// TIA Portal V18 export
TYPE "KukaRobot_UserOutput_3"
   STRUCT
      Public : Struct
         GO_CurrentMode : USInt;
         GO_CurrentPartType : USInt;
         GO_SpeedActual : USInt;   // Robot speed
         GO_RobotTaskSequence : Byte;
         GO5_RobGrip1Status : Byte;   // Gripper 1 status
         GO6_RobGrip2Status : Byte;   // Gripper 2 state
         GO7_Pallet1Count : Byte;
         GO8_UnloadingPalletCount : Byte;   // Pallet finished product count
         GO9 : Byte;
         GO10 : Byte;
      END_STRUCT;
      Gripper : Struct
         DO129_Grip1GoWork : Bool;   // Clamp 1 goes to work position
         DO130_Grip1GoHome : Bool;   // Clamp 1 to original position
         DO131_Grip2GoWork : Bool;   // Clamp 2 goes to work position
         DO132_Grip2GoHome : Bool;   // Clamp 2 to original position
         DO133 : Bool;
         DO134 : Bool;
         DO135 : Bool;
         DO136 : Bool;
         DO137 : Bool;
         DO138 : Bool;
         DO139 : Bool;
         DO140 : Bool;
         DO141 : Bool;
         DO142 : Bool;
         DO143 : Bool;
         DO144 : Bool;
         DO145 : Bool;
         DO146 : Bool;
         DO147 : Bool;
         DO148 : Bool;
         DO149 : Bool;
         DO150 : Bool;
         DO151 : Bool;
         DO152 : Bool;
         DO153 : Bool;
         DO154 : Bool;
         DO155 : Bool;
         DO156 : Bool;
         DO157 : Bool;
         DO158 : Bool;
         DO159 : Bool;
         DO160 : Bool;
      END_STRUCT;
      Home : Struct
         DO161_WaitForHomeSeqStart : Bool;   // The robot waits for the command to be initialized
         DO162_GoHomeFail : Bool;   // The robot fails to automatically return to Home
         DO163_HomeSeqOK : Bool;   // Robot initialization completed
         DO164_WaitForAutoStart : Bool;   // Robot waiting can automatically loop commands
         DO165_AutoCycle : Bool;   // Robot automatic program loop
         DO166 : Bool;
         DO167 : Bool;
         DO168 : Bool;
         DO169 : Bool;
         DO170 : Bool;
         DO171 : Bool;
         DO172 : Bool;
         DO173 : Bool;
         DO174 : Bool;
         DO175 : Bool;
         DO176 : Bool;
         DO177_PressPut1Area : Bool;   // Press installation safety area (0 inside, 1 outside)
         DO178_Robot2Area : Bool;   // Robot 2 safety zone (0 inside, 1 outside)
         DO179_BufferArea : Bool;   // Buffer safe area
         DO180_TableArea : Bool;   // Carousel retrieval safety area
         DO181 : Bool;
         DO182 : Bool;
         DO183 : Bool;
         DO184 : Bool;
         DO185 : Bool;
         DO186 : Bool;
         DO187 : Bool;
         DO188 : Bool;
         DO189 : Bool;
         DO190 : Bool;
         DO191 : Bool;
         DO192 : Bool;
      END_STRUCT;
      Special : Struct
         DO193 : Bool;
         DO194 : Bool;
         DO195 : Bool;
         DO196 : Bool;
         DO197 : Bool;
         DO198 : Bool;
         DO199 : Bool;
         DO200 : Bool;
         DO201 : Bool;
         DO202 : Bool;
         DO203 : Bool;
         DO204 : Bool;
         DO205 : Bool;
         DO206 : Bool;
         DO207 : Bool;
         DO208 : Bool;
         DO209 : Bool;
         DO210 : Bool;
         DO211 : Bool;
         DO212 : Bool;
         DO213 : Bool;
         DO214 : Bool;
         DO215 : Bool;
         DO216 : Bool;
         DO217 : Bool;
         DO218 : Bool;
         DO219 : Bool;
         DO220 : Bool;
         DO221 : Bool;
         DO222 : Bool;
         DO223 : Bool;
         DO224 : Bool;
      END_STRUCT;
      Cycle : Struct
         DO225_ScanPosInside : Bool;   // During tool scanning process
         DO226_ScanPos1Reach : Bool;   // The robot reaches the tool scanning 1 position
         DO227_ScanPos2Reach : Bool;   // The robot reaches the tool scanning 2 position
         DO228_ScanPos3Reach : Bool;   // The robot reaches position 3 of tool scanning code
         DO229_ScanPos4Reach : Bool;   // The robot reaches position 4 of tool scanning code
         DO230_ScanPos5Reach : Bool;   // The robot reaches position 5 of tool scanning code
         DO231_ScanPos6Reach : Bool;   // The robot reaches position 6 of the tool scan code
         DO232_ScanPos7Reach : Bool;   // The robot reaches position 7 of the workwear scan code
         DO233_ScanPoseFinish : Bool;   // Workwear scan completed
         DO234 : Bool;
         DO235 : Bool;
         DO236 : Bool;
         DO237 : Bool;
         DO238 : Bool;
         DO239 : Bool;
         DO240 : Bool;
         DO241_PickPalletInside : Bool;
         DO242_PickPalletFinish : Bool;
         DO243_PickPalletFull : Bool;
         DO244 : Bool;
         DO245 : Bool;
         DO246 : Bool;
         DO247 : Bool;
         DO248 : Bool;
         DO249_PickMagnetInside : Bool;   // Magnet NG in the process of picking up materials
         DO250_PickMagnetFinish : Bool;   // Magnet NG material retrieval completed
         DO251 : Bool;
         DO252 : Bool;
         DO253_PickGlueNGInside : Bool;   // During the process of dispensing NG materials
         DO254_PickGlueNGFinish : Bool;   // Dispensing NG material retrieval completed
         DO255 : Bool;
         DO256 : Bool;
         DO257_PickTableInside : Bool;   // During the turntable retrieval process, 2# area small turntable
         DO258_PickTableFinish : Bool;   // Turntable retrieval completed
         DO259 : Bool;
         DO260 : Bool;
         DO261_ScanRingtInside : Bool;   // Ring scanning process
         DO262_ScanRingFinish : Bool;   // Ring scan completed
         DO263_ScanReach : Bool;   // Scan the code to reach the signal
         DO264 : Bool;
         DO265_LoadNGInside : Bool;   // During NG discharging process
         DO266_LoadNGFinish : Bool;   // NG discharge completed
         DO267 : Bool;
         DO268 : Bool;
         DO269 : Bool;
         DO270 : Bool;
         DO271 : Bool;
         DO272 : Bool;
         DO273_PressPutPart1Inside : Bool;
         DO274_PressPutPart1Finish : Bool;
         DO275 : Bool;
         DO276 : Bool;
         DO277_PressPutRingInside : Bool;   // During the discharging process of press-fitting Ring
         DO278_PressPutRingFinish : Bool;   // Press-mounted Ring discharging completed
         DO279_Press2Reach : Bool;
         DO280 : Bool;
         DO281_PressPickInside : Bool;   // During the press loading and picking process
         DO282_PressPickFinish : Bool;   // Pressing and loading completed
         DO283 : Bool;
         DO284 : Bool;
         DO285 : Bool;
         DO286 : Bool;
         DO287 : Bool;
         DO288 : Bool;
         DO289_PutOkPartInside : Bool;   // During the unloading process of finished parts
         DO290_PutOkPartFinish : Bool;   // Finished parts blanking completed
         DO291_PutPalletFull : Bool;   // Finished parts are fully loaded
         DO292 : Bool;
         DO293 : Bool;
         DO294 : Bool;
         DO295 : Bool;
         DO296 : Bool;
         DO297_MaintainInside : Bool;
         DO298_MaintainFinish : Bool;
         DO299 : Bool;
         DO300_HomeInside : Bool;
         DO301_HomeFinish : Bool;
         DO302 : Bool;
         DO303 : Bool;
         DO304 : Bool;
         DO305_GripScanInside : Bool;
         DO306_GripScanFinish : Bool;
         DO307_ScanPos1Reach : Bool;
         DO308_ScanPos2Reach : Bool;
         DO309_ScanPos3Reach : Bool;
         DO310_ScanPos4Reach : Bool;
         DO311 : Bool;
         DO312 : Bool;
         DO313 : Bool;
         DO314 : Bool;
         DO315 : Bool;
         DO316 : Bool;
         DO317 : Bool;
         DO318 : Bool;
         DO319 : Bool;
         DO320 : Bool;
         DO321 : Bool;
         DO322 : Bool;
         DO323 : Bool;
         DO324 : Bool;
         DO325 : Bool;
         DO326 : Bool;
         DO327 : Bool;
         DO328 : Bool;
         DO329 : Bool;
         DO330 : Bool;
         DO331 : Bool;
         DO332 : Bool;
         DO333 : Bool;
         DO334 : Bool;
         DO335 : Bool;
         DO336 : Bool;
         DO337 : Bool;
         DO338 : Bool;
         DO339 : Bool;
         DO340 : Bool;
         DO341 : Bool;
         DO342 : Bool;
         DO343 : Bool;
         DO344 : Bool;
         DO345 : Bool;
         DO346 : Bool;
         DO347 : Bool;
         DO348 : Bool;
         DO349 : Bool;
         DO350 : Bool;
         DO351 : Bool;
         DO352 : Bool;
         DO353 : Bool;
         DO354 : Bool;
         DO355 : Bool;
         DO356 : Bool;
         DO357 : Bool;
         DO358 : Bool;
         DO359 : Bool;
         DO360 : Bool;
         DO361 : Bool;
         DO362 : Bool;
         DO363 : Bool;
         DO364 : Bool;
         DO365 : Bool;
         DO366 : Bool;
         DO367 : Bool;
         DO368 : Bool;
         DO369 : Bool;
         DO370 : Bool;
         DO371 : Bool;
         DO372 : Bool;
         DO373 : Bool;
         DO374 : Bool;
         DO375 : Bool;
         DO376 : Bool;
         DO377 : Bool;
         DO378 : Bool;
         DO379 : Bool;
         DO380 : Bool;
         DO381 : Bool;
         DO382 : Bool;
         DO383 : Bool;
         DO384 : Bool;
         DO385 : Bool;
         DO386 : Bool;
         DO387 : Bool;
         DO388 : Bool;
         DO389 : Bool;
         DO390 : Bool;
         DO391 : Bool;
         DO392 : Bool;
         DO393 : Bool;
         DO394 : Bool;
         DO395 : Bool;
         DO396 : Bool;
         DO397 : Bool;
         DO398 : Bool;
         DO399 : Bool;
         DO400 : Bool;
         DO401 : Bool;
         DO402 : Bool;
         DO403 : Bool;
         DO404 : Bool;
         DO405 : Bool;
         DO406 : Bool;
         DO407 : Bool;
         DO408 : Bool;
         DO409 : Bool;
         DO410 : Bool;
         DO411 : Bool;
         DO412 : Bool;
         DO413 : Bool;
         DO414 : Bool;
         DO415 : Bool;
         DO416 : Bool;
      END_STRUCT;
      Safety : Struct
         DO417 : Bool;
         DO418 : Bool;
         DO419 : Bool;
         DO420 : Bool;
         DO421 : Bool;
         DO422 : Bool;
         DO423 : Bool;
         DO424 : Bool;
         DO425 : Bool;
         DO426 : Bool;
         DO427 : Bool;
         DO428 : Bool;
         DO429 : Bool;
         DO430 : Bool;
         DO431 : Bool;
         DO432 : Bool;
         DO433 : Bool;
         DO434 : Bool;
         DO435 : Bool;
         DO436 : Bool;
         DO437 : Bool;
         DO438 : Bool;
         DO439 : Bool;
         DO440 : Bool;
         DO441 : Bool;
         DO442 : Bool;
         DO443 : Bool;
         DO444 : Bool;
         DO445 : Bool;
         DO446 : Bool;
         DO447 : Bool;
         DO448 : Bool;
         DO449 : Bool;
         DO450 : Bool;
         DO451 : Bool;
         DO452 : Bool;
         DO453 : Bool;
         DO454 : Bool;
         DO455 : Bool;
         DO456 : Bool;
         DO457 : Bool;
         DO458 : Bool;
         DO459 : Bool;
         DO460 : Bool;
         DO461 : Bool;
         DO462 : Bool;
         DO463 : Bool;
         DO464 : Bool;
         DO465 : Bool;
         DO466 : Bool;
         DO467 : Bool;
         DO468 : Bool;
         DO469 : Bool;
         DO470 : Bool;
         DO471 : Bool;
         DO472 : Bool;
         DO473 : Bool;
         DO474 : Bool;
         DO475 : Bool;
         DO476 : Bool;
         DO477 : Bool;
         DO478 : Bool;
         DO479 : Bool;
         DO480 : Bool;
         DO481 : Bool;
         DO482 : Bool;
         DO483 : Bool;
         DO484 : Bool;
         DO485 : Bool;
         DO486 : Bool;
         DO487 : Bool;
         DO488 : Bool;
         DO489 : Bool;
         DO490 : Bool;
         DO491 : Bool;
         DO492 : Bool;
         DO493 : Bool;
         DO494 : Bool;
         DO495 : Bool;
         DO496 : Bool;
         DO497 : Bool;
         DO498 : Bool;
         DO499 : Bool;
         DO500 : Bool;
         DO501 : Bool;
         DO502 : Bool;
         DO503 : Bool;
         DO504 : Bool;
         DO505 : Bool;
         DO506 : Bool;
         DO507 : Bool;
         DO508 : Bool;
         DO509 : Bool;
         DO510 : Bool;
         DO511 : Bool;
         DO512 : Bool;
      END_STRUCT;
   END_STRUCT;
END_TYPE
